FUNCTION_BLOCK TRAFFICLIGHT_HMI (* Hmi for one set of traffic lights *)
  (* Standard: 61499-1; Classification: HMI; Function: Output; Type: 4xLED *)
  (* Version 0.3, 2011-03-28, JHC, Holobloc Inc, Updated documentation. *)
  (* Version 0.2, 2008-11-10, JHC, Holobloc Inc, Moved to fb.rt.doc. *)
  (* Version 0.1, 2008-06-04, JHC, Holobloc Inc, Updated DOCTYPE. *)
  (* Version 0.0, 2001-02-21, JHC, Rockwell Automation *)
  (* Compiler header: package fb.rt.dasdA1; import fb.rt.hmi.*; *)
  (* Compiler Java Sun JDK 1.6.0 *)
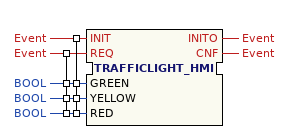
  EVENT_INPUT
    INIT WITH GREEN, YELLOW, RED; (* Initialization Request *)
    REQ WITH GREEN, YELLOW, RED; (* Display Request *)
  END_EVENT
  EVENT_OUTPUT
    INITO; (* Initialization Confirm *)
    CNF; (* Execution Confirmation *)
  END_EVENT
  VAR_INPUT
    GREEN : BOOL;
    YELLOW : BOOL;
    RED : BOOL;
  END_VAR
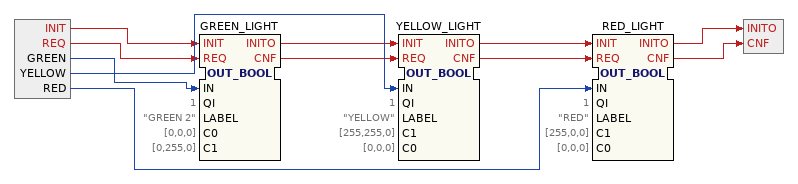
  FBS
    GREEN_LIGHT : OUT_BOOL(QI := 1, LABEL := "GREEN 2", C0 := [0,0,0], C1 := [0,255,0]);
    YELLOW_LIGHT : OUT_BOOL(QI := 1, LABEL := "YELLOW", C1 := [255,255,0], C0 := [0,0,0]);
    RED_LIGHT : OUT_BOOL(QI := 1, LABEL := "RED", C1 := [255,0,0], C0 := [0,0,0]);
  END_FBS
  EVENT_CONNECTIONS
    GREEN_LIGHT.INITO TO YELLOW_LIGHT.INIT;
    YELLOW_LIGHT.INITO TO RED_LIGHT.INIT;
    RED_LIGHT.INITO TO INITO;
    GREEN_LIGHT.CNF TO YELLOW_LIGHT.REQ;
    YELLOW_LIGHT.CNF TO RED_LIGHT.REQ;
    RED_LIGHT.CNF TO CNF;
    INIT TO GREEN_LIGHT.INIT;
    REQ TO GREEN_LIGHT.REQ;
  END_CONNECTIONS
  DATA_CONNECTIONS
    GREEN TO GREEN_LIGHT.IN;
    YELLOW TO YELLOW_LIGHT.IN;
    RED TO RED_LIGHT.IN;
  END_CONNECTIONS
END_FUNCTION_BLOCK
